{attribute 'OPC.UA.DA.JobMethod' := 'JobMethode_RotationMove'}
FUNCTION_BLOCK VSG_AS_RotationMoveEncoder
VAR
	AlwaysTrue : BOOL := TRUE;
	// Used for debugging purposes to display InputArguments of method call
	MethodCall_RotationMove : BOOL := FALSE; // used to store InputArg "MethodCall" from Start() method
	Direction : BOOL := FALSE;
	EncoderTargetPosition_01 : BOOL;
	EncoderTargetPosition_02 : BOOL;
	callCounterStart : ULINT; // counts how many times the Start() method has been called
	callCounterCheckState : ULINT; // counts how many times the CheckState() method has been called
	callCounterAbort : ULINT; // counts how many times the Abort() method has been called
	
	// Variables to determine if a job has been started (Start() method has been called) or finished
	jobRunning : BOOL;
	jobFinished : BOOL;

	// State machine variable
	state : UDINT;
	
	//Variablen des Transport FBs
	ResetCall	: BOOL := FALSE;
	HRL_RGB_VerticalMoveWithEncoder : AxisControl_Encoder;
END_VAR
	
VAR_INPUT
	NotAusSignal: BOOL;
	EncoderStartPosition_01 : BOOL;
	EncoderStartPosition_02 : BOOL;
//	TOF_Time_Motoransteuerung : TIME;
//	TOF_Time_EndschalterEntlastung : TIME;
END_VAR

VAR_OUTPUT
	Motor_Ansteuerung01 : BOOL;
	Motor_Ansteuerung02 : BOOL;
END_VAR

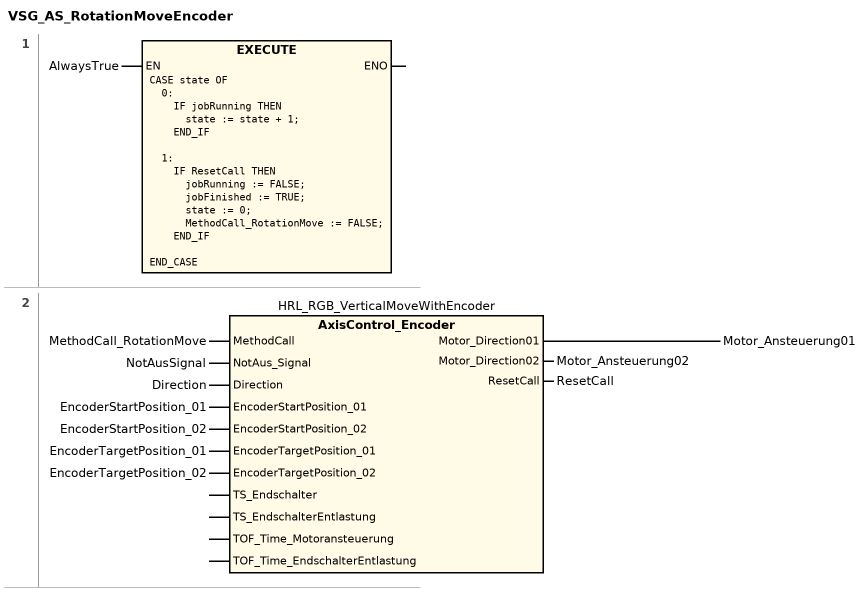
// NETWORK 1
IF AlwaysTrue THEN
    CASE state OF
    	0:
    		IF jobRunning THEN
    			state := state + 1;
    		END_IF
    		
    	1:
    		IF ResetCall THEN
    			jobRunning := FALSE;
    			jobFinished := TRUE;
    			state := 0;
    			MethodCall_RotationMove := FALSE;
    		END_IF
    		
    END_CASE
END_IF

// NETWORK 2
HRL_RGB_VerticalMoveWithEncoder(
    MethodCall := MethodCall_RotationMove,
    NotAus_Signal := NotAusSignal,
    Direction := Direction,
    EncoderStartPosition_01 := EncoderStartPosition_01,
    EncoderStartPosition_02 := EncoderStartPosition_02,
    EncoderTargetPosition_01 := EncoderTargetPosition_01,
    EncoderTargetPosition_02 := EncoderTargetPosition_02,
    Motor_Direction02 => Motor_Ansteuerung02,
    ResetCall => ResetCall); // AxisControl_Encoder
Motor_Ansteuerung01 := HRL_RGB_VerticalMoveWithEncoder.Motor_Direction01;

{attribute 'TcRpcEnable' := '1'}
METHOD Abort : HRESULT
VAR_INPUT
	hdl : UDINT; // Do not change, used by server.
END_VAR
callCounterAbort := callCounterAbort + 1;
END_METHOD

{attribute 'TcRpcEnable' := '1'}
METHOD CheckState : HRESULT
VAR_INPUT
	hdl : UDINT; // Do not change, used by server.
END_VAR
VAR_OUTPUT
	bBusy : BOOL; // Do not change. Used by server to find out if the job is finished
	
	// List of OutputArguments for OPC UA method, may be customized
	State : BOOL; // Abgeschlossener MethodCall
	MethodCall: BOOL; //Input Recall
END_VAR
callCounterCheckState := callCounterCheckState + 1;
IF NOT jobFinished THEN
	bBusy := TRUE; // job is not finished yet
	CheckState := 0; // no error
ELSE
	bBusy := FALSE; // job is finished
	CheckState := 0; // done, no error occured during execution (OPC UA StatusCode "GOOD")
	jobFinished := FALSE;
	State := ResetCall;
	MethodCall := MethodCall_RotationMove;
END_IF
END_METHOD

{attribute 'TcRpcEnable' := '1'}
METHOD Start : HRESULT
VAR_INPUT
	// List of InputArguments for OPC UA method, may be customized
	MethodCall : BOOL; // some description
	DirectionPoint : BOOL;
	EncoderPositionVertical_01 : BOOL;
	EncoderPositionVertical_02 : BOOL;
END_VAR
VAR_OUTPUT
	hdl : UDINT; // Do not change, used by server.
END_VAR
callCounterStart := callCounterStart + 1;

MethodCall_RotationMove := MethodCall;
DirectionPoint := Direction;
EncoderTargetPosition_01 := EncoderPositionVertical_01;
EncoderTargetPosition_02 := EncoderPositionVertical_02;

jobRunning := TRUE;
Start := 0; // no error occured, e.g. while parsing the input arguments (0 = OPC UA StatusCode "GOOD")
END_METHOD

END_FUNCTION_BLOCK

(* stored: Version 1.1.0.1, ProductVersion 3.1.4024.15
   POU VSG_AS_RotationMoveEncoder: Id {79321839-ea1c-4ef0-b797-4ae15528adb2}, SpecialFunc None
   Method Abort: Id {97b0e0a6-e20c-4469-9650-bdbea8d06504}
   Method CheckState: Id {2f628288-7258-4536-8831-c80322f1cd2d}
   Method Start: Id {4e3c69c1-cb4f-4b2b-b8c6-3088c729869c} *)
